{attribute addProperty BoxType "EL1259-0000-0016"}
{attribute addProperty Id "Output_short_circuitBIT10.1251Output_buffer_overflowBIT10.1252Output_stateBIT10.1253Input_cycle_counter_BIT_0BIT10.12515Input_cycle_counter_BIT_1BIT10.12515Output_order_feedbackUSINT8117Events_in_output_bufferUSINT8118"}
{attribute addProperty CRC "850971234"}
{attribute addProperty SizeInBites "109"}
{attribute addProperty SizeInBytes "13.625"}
{warning 'Size of this structure is not a multiple of 8 bits!!!'}
TYPE Status_32B8CA62 :
STRUCT
	{attribute addProperty Name "Output_short_circuit"}
	Output_short_circuit : BIT;
	{attribute addProperty Name "Output_buffer_overflow"}
	Output_buffer_overflow : BIT;
	{attribute addProperty Name "Output_state"}
	Output_state : BIT;
	{attribute 'hide'}
	reserve_1_BOOL_0 : BOOL;
	{attribute 'hide'}
	reserve_1_BOOL_1 : BOOL;
	{attribute 'hide'}
	reserve_1_BOOL_2 : BOOL;
	{attribute 'hide'}
	reserve_1_BOOL_3 : BOOL;
	{attribute 'hide'}
	reserve_1_BOOL_4 : BOOL;
	{attribute 'hide'}
	reserve_1_BOOL_5 : BOOL;
	{attribute 'hide'}
	reserve_1_BOOL_6 : BOOL;
	{attribute 'hide'}
	reserve_1_BOOL_7 : BOOL;
	{attribute 'hide'}
	reserve_1_BOOL_8 : BOOL;
	{attribute 'hide'}
	reserve_1_BOOL_9 : BOOL;
	{attribute 'hide'}
	reserve_1_BOOL_10 : BOOL;
	{attribute addProperty Name "Input_cycle_counter"}
	Input_cycle_counter_BIT_0 : BIT;
	{attribute addProperty Name "Input_cycle_counter"}
	Input_cycle_counter_BIT_1 : BIT;
	{attribute addProperty Name "Output_order_feedback"}
	Output_order_feedback : USINT;
	{attribute addProperty Name "Events_in_output_buffer"}
	Events_in_output_buffer : USINT;
END_STRUCT
END_TYPE

(* stored: Version 1.2.0.0, ProductVersion 3.1.4024.9
   DUT Status_32B8CA62: Id {84238114-982a-4ceb-b9ad-9882d3fcc07e} *)
